FUNCTION_BLOCK FB_ResetDescargador_SFC

VAR_INPUT
	//nuestras_variables

    // SFC-Flags
    SFCPause: BOOL;
    SFCReset: BOOL;
    
    // Indicadores de sincronizacion
    Ack: BOOL := TRUE;
    Execute: BOOL;
	
	//Entradas
    Horizontal_descargador_detras: BOOL;
	Vertical_descargador_arriba: BOOL;

	
END_VAR
VAR_OUTPUT
    // Indicadores de sincronizacion
    Done: BOOL;
    Ready: BOOL;

	//Salidas
	Descargador_atras: BOOL;
	
END_VAR
VAR
END_VAR

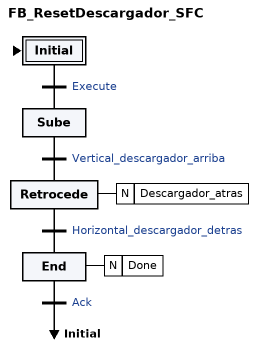
INITIAL_STEP Initial:
END_STEP
TRANSITION FROM Initial TO Sube
    := Execute;
END_TRANSITION
STEP Sube:
END_STEP
TRANSITION FROM Sube TO Retrocede
    := Vertical_descargador_arriba;
END_TRANSITION
STEP Retrocede:
    Descargador_atras(N);
END_STEP
TRANSITION FROM Retrocede TO End
    := Horizontal_descargador_detras;
END_TRANSITION
STEP End:
    Done(N);
END_STEP
TRANSITION FROM End TO Initial
    := Ack;
END_TRANSITION

END_FUNCTION_BLOCK

(* stored: Version 1.1.0.1, ProductVersion 3.1.4024.12
   POU FB_ResetDescargador_SFC: Id {93829831-eb30-4810-992a-71b04d0a49a1}, SpecialFunc None *)
